// TIA Portal project "TaslamaTezgahiUygulamasi" (V17)

(* hardware
DEVICE "S7-1200 station_1"  S7-1200 Station
   slot 0: "Rack_0"  S7-1200 Rack  Rack  V1.0
   slot 1: "PLC_1"  CPU 1214C DC/DC/DC  6ES7 214-1AG40-0XB0  V4.5
*)

// ===== PLC "PLC_1"  CPU 1214C DC/DC/DC =====

VAR_GLOBAL   // PLC tag table "Default tag table"
   "TAŞ MOTORU" AT %Q0.0 : Bool;
   "POMPA KAPAMA BUTONU" AT %I0.0 : Bool;
   "POMPA MOTORU" AT %Q0.1 : Bool;
   "POMPA AÇMA BUTONU" AT %I0.1 : Bool;
   "TAŞ KAPAMA BUTONU" AT %I0.2 : Bool;
   "TERMİK SİGORTA" AT %I0.3 : Bool;
   "TAŞ AÇMA BUTONU" AT %I0.4 : Bool;
END_VAR

ORGANIZATION_BLOCK "Main"   // OB1, LAD, ProgramCycle
TITLE = "Main Program Sweep (Cycle)"
{ S7_Optimized_Access := 'TRUE' }
VERSION : 0.1
   VAR_INPUT
      Initial_Call : Bool;   // Initial call of this OB
      Remanence : Bool;   // =True, if remanent data are available
   END_VAR
BEGIN

REGION Network 1: POMPANIN ÇALIŞMASI
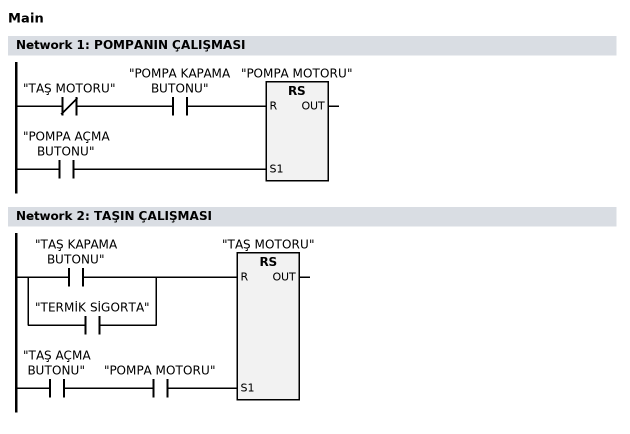
   RUNG wire#powerrail
      I_Contact( "TAŞ MOTORU" )
      Contact( "POMPA KAPAMA BUTONU" )
      S_RS(operand := "POMPA MOTORU", s1 := wire#w1)
   END_RUNG
   RUNG wire#powerrail
      Contact( "POMPA AÇMA BUTONU" )
   END_RUNG wire#w1
   // the same network as SCL:
   IF NOT "TAŞ MOTORU" AND "POMPA KAPAMA BUTONU" THEN
       "POMPA MOTORU" := FALSE;   // RS flip-flop
   END_IF;
   IF "POMPA AÇMA BUTONU" THEN "POMPA MOTORU" := TRUE; END_IF;
END_REGION

REGION Network 2: TAŞIN ÇALIŞMASI
   RUNG wire#powerrail
      Contact( "TAŞ KAPAMA BUTONU" )
      wire#w1
      S_RS(operand := "TAŞ MOTORU", s1 := wire#w2)
   END_RUNG
   RUNG wire#powerrail
      Contact( "TERMİK SİGORTA" )
   END_RUNG wire#w1
   RUNG wire#powerrail
      Contact( "TAŞ AÇMA BUTONU" )
      Contact( "POMPA MOTORU" )
   END_RUNG wire#w2
   // the same network as SCL:
   IF "TAŞ KAPAMA BUTONU" OR "TERMİK SİGORTA" THEN
       "TAŞ MOTORU" := FALSE;   // RS flip-flop
   END_IF;
   IF "TAŞ AÇMA BUTONU" AND "POMPA MOTORU" THEN "TAŞ MOTORU" := TRUE; END_IF;
END_REGION
END_ORGANIZATION_BLOCK